(* IEC 61131-3 sources: Std_PalletMover/Class/AutomaticControl, 1 file *)

(* ---- AutomaticControl.st ---- *)
(*!
<Class
	Name               = "AutomaticControl"
	Revision           = "0.0"
	RealtimeTask       = "false"
	CyclicTask         = "false"
	BackgroundTask     = "false"
	Sigmatek           = "false"
	OSInterface        = "false"
	HighPriority       = "false"
	Automatic          = "false"
	UpdateMode         = "Prescan"
	SharedCommandTable = "true"
	Objectsize         = "(366,120)">
	<Channels>
		<Server Name="ClassSvr" Visualized="false" Initialize="false" WriteProtected="true" Retentive="false"/>
	</Channels>
</Class>
*)
AutomaticControl : CLASS
	TYPE
#pragma pack(push, 1)
	  tAutomaticControlData : STRUCT  //! <Type Public="true" Name="tAutomaticControlData"/>
	    acd_DrivingVectorAngle : REAL;
	    acd_SteeringRadius : REAL;
	    acd_DrivingSpeed : REAL;
	  END_STRUCT;
#pragma pack(pop)
	END_TYPE
  //Servers:
	ClassSvr 	: SvrChCmd_DINT;
  //Clients:
  //Variables:
  //Functions:

	FUNCTION VIRTUAL GLOBAL SetData
		VAR_INPUT
			data 	: tAutomaticControlData;
		END_VAR;
  //Tables:
	FUNCTION @STD
		VAR_OUTPUT
			ret_code	: CONFSTATES;
		END_VAR;
	FUNCTION GLOBAL TAB @CT_;
END_CLASS;

FUNCTION VIRTUAL GLOBAL AutomaticControl::SetData
  #pragma warning(disable: 73);
  #pragma warning(disable: 76);
	VAR_INPUT
		data 	: tAutomaticControlData;
	END_VAR
  #pragma warning(default: 73);
  #pragma warning(default: 76);
END_FUNCTION
